INTERFACE I_Module

PROPERTY AccessModuleName : String
GET
END_GET
SET
END_SET
END_PROPERTY

END_INTERFACE

(* stored: Version 1.1.0.1, ProductVersion 3.1.4022.16
   Itf I_Module: Id {f00a0672-edfb-4485-859b-c480ea244f69}
   Property AccessModuleName: Id {b3ee3530-aa25-49fe-b0de-5dfaf98beb46}
   Get Get: Id {41360fad-073a-4389-9781-eb3b8b14ecec}
   Set Set: Id {f1fb4c81-ec1e-40ec-aa1d-906060691271} *)
